// TIA Portal V18 export
FUNCTION_BLOCK "mot_speed_wdir_slowly_accelerated"   // FB68, FBD
{ S7_Optimized_Access := 'TRUE' }
VERSION : 0.1
// stored: AutoNumber true, IsIECCheckEnabled false, IsRetainMemResEnabled false, MemoryReserve 100, SetENOAutomatically false, UDAEnableTagReadback false
   VAR_INPUT
      ALLOWED : Bool;
      set_speed__wdir : Real;
      v_absMax : Real;
      t_acc : Real;
      STOP_NOW : Bool;
   END_VAR
   VAR_OUTPUT
      speed_accelerated_slowly_wdir : Real;
   END_VAR
   VAR
      speed_is_zero : Bool;
      speed_is_zero_was : Bool;
      speed_is_zero_CLK : Bool;
   END_VAR
   VAR_TEMP
      cycle_time_s : Real;
      acceleration : Real;
      accleration_per_cycle : Real;
   END_VAR
BEGIN

REGION Network 2 (SCL)
   #speed_is_zero := #set_speed__wdir = 0;
   #speed_is_zero_CLK := false;//AND #speed_is_zero AND NOT #speed_is_zero_was; 
   #speed_is_zero_was := #speed_is_zero ;
END_REGION

REGION Network 3 (SCL)
   #cycle_time_s := "_MAIN_DB".CLOCK_S_P_SCAN;
   IF #t_acc > 0 AND NOT #STOP_NOW THEN
       #acceleration := #v_absMax / #t_acc;
       #accleration_per_cycle := #acceleration * #cycle_time_s;
       IF NOT #ALLOWED OR #speed_is_zero_CLK  THEN
           #speed_accelerated_slowly_wdir := #set_speed__wdir;
       ELSE
           IF #speed_accelerated_slowly_wdir < #set_speed__wdir THEN
               #speed_accelerated_slowly_wdir := MIN(IN1 := #speed_accelerated_slowly_wdir + #accleration_per_cycle, IN2 := #set_speed__wdir);
           ELSE 
               #speed_accelerated_slowly_wdir := MAX(IN1 := #speed_accelerated_slowly_wdir - #accleration_per_cycle,IN2 := #set_speed__wdir);
           END_IF;
       END_IF;
   ELSE
       #speed_accelerated_slowly_wdir := #set_speed__wdir;
   END_IF;
END_REGION
END_FUNCTION_BLOCK
